// Mitsubishi GX Works2 project: GX_GROUP5   PLC: FX3G

// global labels: Global1
VAR_GLOBAL CONSTANT
  reset1 : INT;
END_VAR
VAR_GLOBAL
  analog_output AT D8282 : INT;
  start_switch AT X007 : BOOL;
  work_light AT Y007 : BOOL;
  emerge_switch AT X005 : BOOL;
  invalid_input AT M7 : BOOL;
  invalid_input_pinuk AT M9 : BOOL;
  petel_begin AT D1102 : REAL;
  petel_current AT D1110 : REAL;
  limon_begin AT D1104 : REAL;
  meyatzev_begin AT D1106 : REAL;
  gummybear_begin AT D1108 : REAL;
  limon_current AT D1112 : REAL;
  meyatzev_current AT D1114 : REAL;
  gummybear_current AT D1116 : REAL;
  start_day AT M0 : BOOL;
  start_icecream AT X001 : BOOL;
  analog_input1 AT D8280 : INT;
  new_analog_input1 AT D1118 : REAL;
END_VAR
VAR_GLOBAL CONSTANT
  convert_input : REAL := 400;
END_VAR
VAR_GLOBAL
  new_analog_input2 AT D1120 : REAL;
  begin_analog_input AT M1 : BOOL;
END_VAR
VAR_GLOBAL CONSTANT
  min_petel : REAL := 280;
  min_limon : REAL := 455;
  min_meyatzev : REAL := 105;
  min_gummybear : REAL := 28;
  const6 : REAL := 6;
  const5 : REAL := 5;
END_VAR
VAR_GLOBAL
  pinuk_ic AT M2 : BOOL;
  regular_ic AT M3 : BOOL;
END_VAR
VAR_GLOBAL CONSTANT
  const385 : REAL := 385;
  const665 : REAL := 665;
  const210 : REAL := 210;
  const70 : REAL := 70;
END_VAR
VAR_GLOBAL
  petelic_container AT D1122 : REAL;
END_VAR
VAR_GLOBAL CONSTANT
  const350 : REAL := 350;
END_VAR
VAR_GLOBAL
  limonic_container AT D1124 : REAL;
END_VAR
VAR_GLOBAL CONSTANT
  const490 : REAL := 490;
END_VAR
VAR_GLOBAL
  finish_regular AT M5 : BOOL;
END_VAR
VAR_GLOBAL CONSTANT
  const560 : REAL := 560;
  const700 : REAL := 700;
END_VAR
VAR_GLOBAL
  finish_pinuk AT M4 : BOOL;
  making_light AT Y000 : BOOL;
  finish_making AT TS1 : BOOL;
  making_time AT TC1 : BOOL;
END_VAR
VAR_GLOBAL CONSTANT
  making_time50 : INT := 50;
  reset_container : REAL;
END_VAR
VAR_GLOBAL
  petel_cooling AT D1126 : REAL;
  limon_cooling AT D1128 : REAL;
  start_cooling AT X002 : BOOL;
  finish_cooling AT Y002 : BOOL;
  sen10 AT X003 : BOOL;
  cooling_timer AT TC2 : BOOL;
END_VAR
VAR_GLOBAL CONSTANT
  cooling_time80 : INT := 80;
END_VAR
VAR_GLOBAL
  container_mix AT D1130 : REAL;
  transfered_to_mix AT M11 : BOOL;
END_VAR
VAR_GLOBAL CONSTANT
  mix_regular_gummybear : REAL := 28;
END_VAR
VAR_GLOBAL
  mix_regular_full AT M12 : BOOL;
  cooling_time AT TS2 : BOOL;
  check AT M101 : BOOL;
  petel_cooling_full AT M10 : BOOL;
  limon_cooling_full AT M17 : BOOL;
END_VAR
VAR_GLOBAL CONSTANT
  mix_pinuk_gummybear : REAL := 70;
END_VAR
VAR_GLOBAL
  mix_pinuk_full AT M13 : BOOL;
  container_mix_total AT D1330 : REAL;
  ready_to_mix AT M15 : BOOL;
END_VAR
VAR_GLOBAL CONSTANT
  regular_mix_time : INT := 30;
END_VAR
VAR_GLOBAL
  mixing_time AT D1132 : INT;
END_VAR
VAR_GLOBAL CONSTANT
  pinuk_mixing_time : INT := 50;
END_VAR
VAR_GLOBAL
  new_mixing_time AT D1134 : INT;
  mixing_time_counter AT TC3 : BOOL;
  finish_counter_mix AT TS3 : BOOL;
  flash_light_mix AT M14 : BOOL;
  flash1 AT TC4 : BOOL;
END_VAR
VAR_GLOBAL CONSTANT
  flash_duration : INT := 5;
END_VAR
VAR_GLOBAL
  timer1 AT TS4 : BOOL;
  light5 AT Y005 : BOOL;
  light6 AT Y006 : BOOL;
  timer2 AT TS5 : BOOL;
  flash2 AT TC5 : BOOL;
  start_packing AT X004 : BOOL;
  first_pack AT CC1 : BOOL;
  counter_pack AT CC2 : BOOL;
  pack_cone AT X000 : BOOL;
END_VAR
VAR_GLOBAL CONSTANT
  counter1 : INT := 1;
END_VAR
VAR_GLOBAL
  outCC2 AT CS2 : BOOL;
  packing AT Y004 : BOOL;
  outCS1 AT CS1 : BOOL;
END_VAR
VAR_GLOBAL CONSTANT
  counter6 : INT := 6;
END_VAR
VAR_GLOBAL
  iteration_help AT M100 : BOOL;
END_VAR
VAR_GLOBAL CONSTANT
  counter7 : INT := 7;
  add_package : INT := 1;
  sec : INT := 10;
END_VAR
VAR_GLOBAL
  amount_packages AT D1200 : REAL;
END_VAR
VAR_GLOBAL CONSTANT
  one_package : REAL := 1;
END_VAR
VAR_GLOBAL
  check2 AT M102 : BOOL;
  finish_making_light AT M200 : BOOL;
  finish_cooling_light AT M201 : BOOL;
END_VAR
VAR_GLOBAL CONSTANT
  const40 : REAL := 40;
END_VAR
VAR_GLOBAL
  new_amount_package AT D1136 : REAL;
END_VAR

// task Task_01 (event TRUE, interval 0, priority 31): POU_01

PROGRAM POU_01
(* structured ladder/FBD written out as ST: instructions are called as NAME(EN, inputs, outputs); _pN, _eN, _tN stand for wires *)
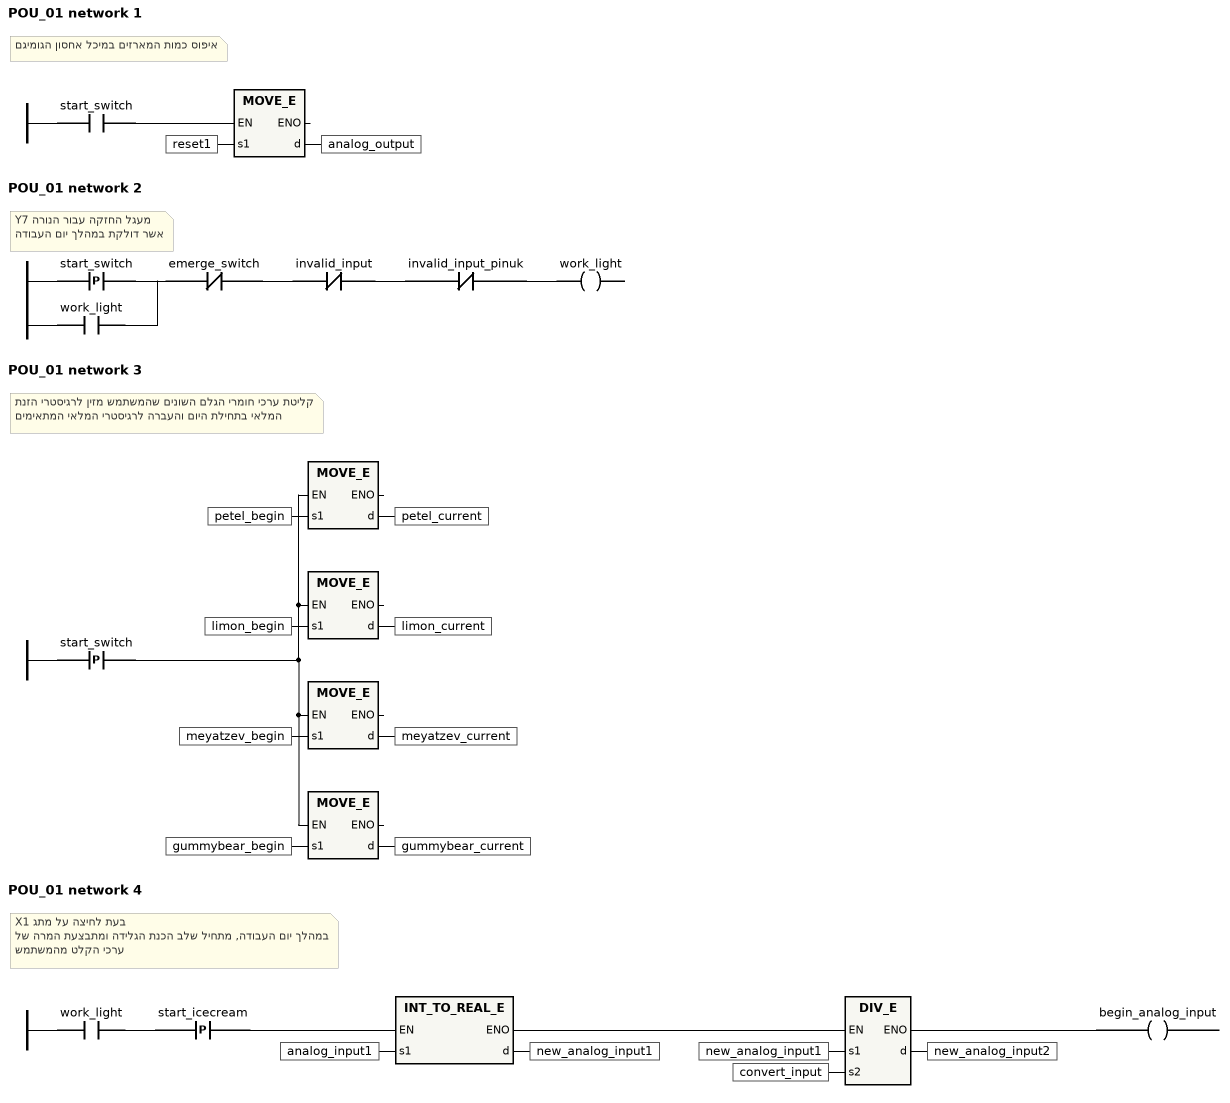
(* network 1 *)
(* איפוס כמות המארזים במיכל אחסון הגומיגם *)
MOVE_E(start_switch, reset1, analog_output);
(* network 2 *)
(* מעגל החזקה עבור הנורה Y7 /  אשר דולקת במהלך יום העבודה *)
work_light := (((LDP(TRUE, start_switch) OR work_light) AND NOT emerge_switch) AND NOT invalid_input) AND NOT invalid_input_pinuk;
(* network 3 *)
(* קליטת ערכי חומרי הגלם השונים שהמשתמש מזין לרגיסטרי הזנת המלאי בתחילת היום והעברה לרגיסטרי המלאי המתאימים *)
_p1 := LDP(TRUE, start_switch);
MOVE_E(_p1, petel_begin, petel_current);
MOVE_E(_p1, limon_begin, limon_current);
MOVE_E(_p1, meyatzev_begin, meyatzev_current);
MOVE_E(_p1, gummybear_begin, gummybear_current);
(* network 4 *)
(* בעת לחיצה על מתג X1  / במהלך יום העבודה, מתחיל שלב הכנת הגלידה ומתבצעת המרה של ערכי הקלט מהמשתמש *)
_e1 := INT_TO_REAL_E(work_light AND LDP(TRUE, start_icecream), analog_input1, new_analog_input1);
_e2 := DIV_E(_e1, new_analog_input1, convert_input, new_analog_input2);
begin_analog_input := _e2;
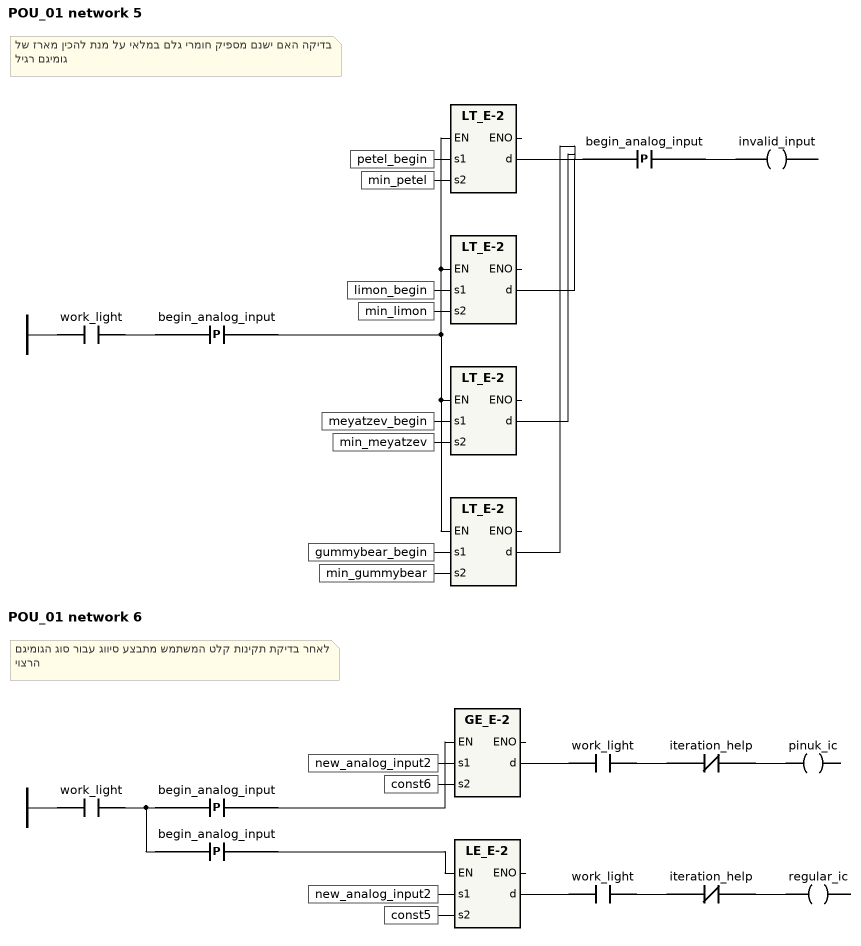
(* network 5 *)
(* בדיקה האם ישנם מספיק חומרי גלם במלאי על מנת להכין מארז של גומיגם רגיל *)
_p1 := work_light AND LDP(TRUE, begin_analog_input);
LT_E(_p1, petel_begin, min_petel, _t2);
LT_E(_p1, limon_begin, min_limon, _t3);
LT_E(_p1, meyatzev_begin, min_meyatzev, _t4);
LT_E(_p1, gummybear_begin, min_gummybear, _t5);
invalid_input := (_t2 OR _t3 OR _t4 OR _t5) AND LDP(TRUE, begin_analog_input);
(* network 6 *)
(* לאחר בדיקת תקינות קלט המשתמש מתבצע סיווג עבור סוג הגומיגם הרצוי *)
GE_E(work_light AND LDP(TRUE, begin_analog_input), new_analog_input2, const6, _t1);
pinuk_ic := _t1 AND work_light AND NOT iteration_help;
LE_E(work_light AND LDP(TRUE, begin_analog_input), new_analog_input2, const5, _t2);
regular_ic := _t2 AND work_light AND NOT iteration_help;
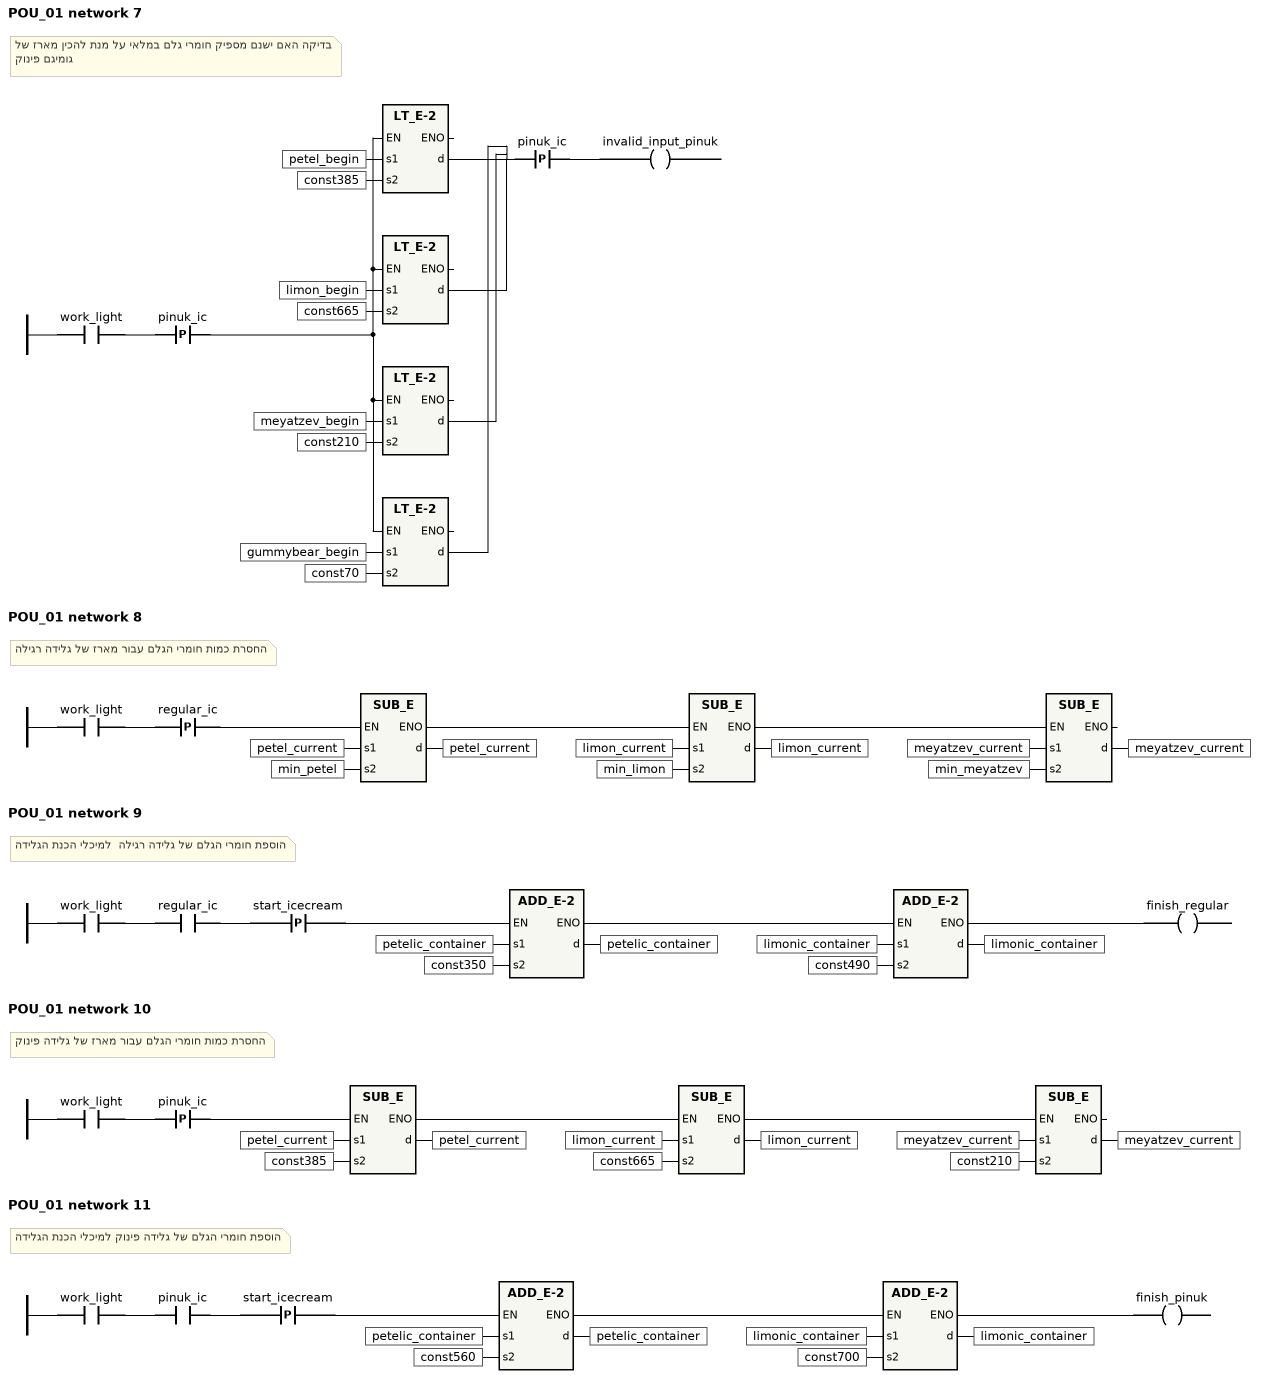
(* network 7 *)
(* בדיקה האם ישנם מספיק חומרי גלם במלאי על מנת להכין מארז של גומיגם פינוק *)
_p1 := work_light AND LDP(TRUE, pinuk_ic);
LT_E(_p1, petel_begin, const385, _t2);
LT_E(_p1, limon_begin, const665, _t3);
LT_E(_p1, meyatzev_begin, const210, _t4);
LT_E(_p1, gummybear_begin, const70, _t5);
invalid_input_pinuk := (_t2 OR _t3 OR _t4 OR _t5) AND LDP(TRUE, pinuk_ic);
(* network 8 *)
(* החסרת כמות חומרי הגלם עבור מארז של גלידה רגילה *)
_e1 := SUB_E(work_light AND LDP(TRUE, regular_ic), petel_current, min_petel, petel_current);
_e2 := SUB_E(_e1, limon_current, min_limon, limon_current);
SUB_E(_e2, meyatzev_current, min_meyatzev, meyatzev_current);
(* network 9 *)
(* הוספת חומרי הגלם של גלידה רגילה  למיכלי הכנת הגלידה *)
_e1 := ADD_E(work_light AND regular_ic AND LDP(TRUE, start_icecream), petelic_container, const350, petelic_container);
_e2 := ADD_E(_e1, limonic_container, const490, limonic_container);
finish_regular := _e2;
(* network 10 *)
(* החסרת כמות חומרי הגלם עבור מארז של גלידה פינוק *)
_e1 := SUB_E(work_light AND LDP(TRUE, pinuk_ic), petel_current, const385, petel_current);
_e2 := SUB_E(_e1, limon_current, const665, limon_current);
SUB_E(_e2, meyatzev_current, const210, meyatzev_current);
(* network 11 *)
(* הוספת חומרי הגלם של גלידה פינוק למיכלי הכנת הגלידה *)
_e1 := ADD_E(work_light AND pinuk_ic AND LDP(TRUE, start_icecream), petelic_container, const560, petelic_container);
_e2 := ADD_E(_e1, limonic_container, const700, limonic_container);
finish_pinuk := _e2;
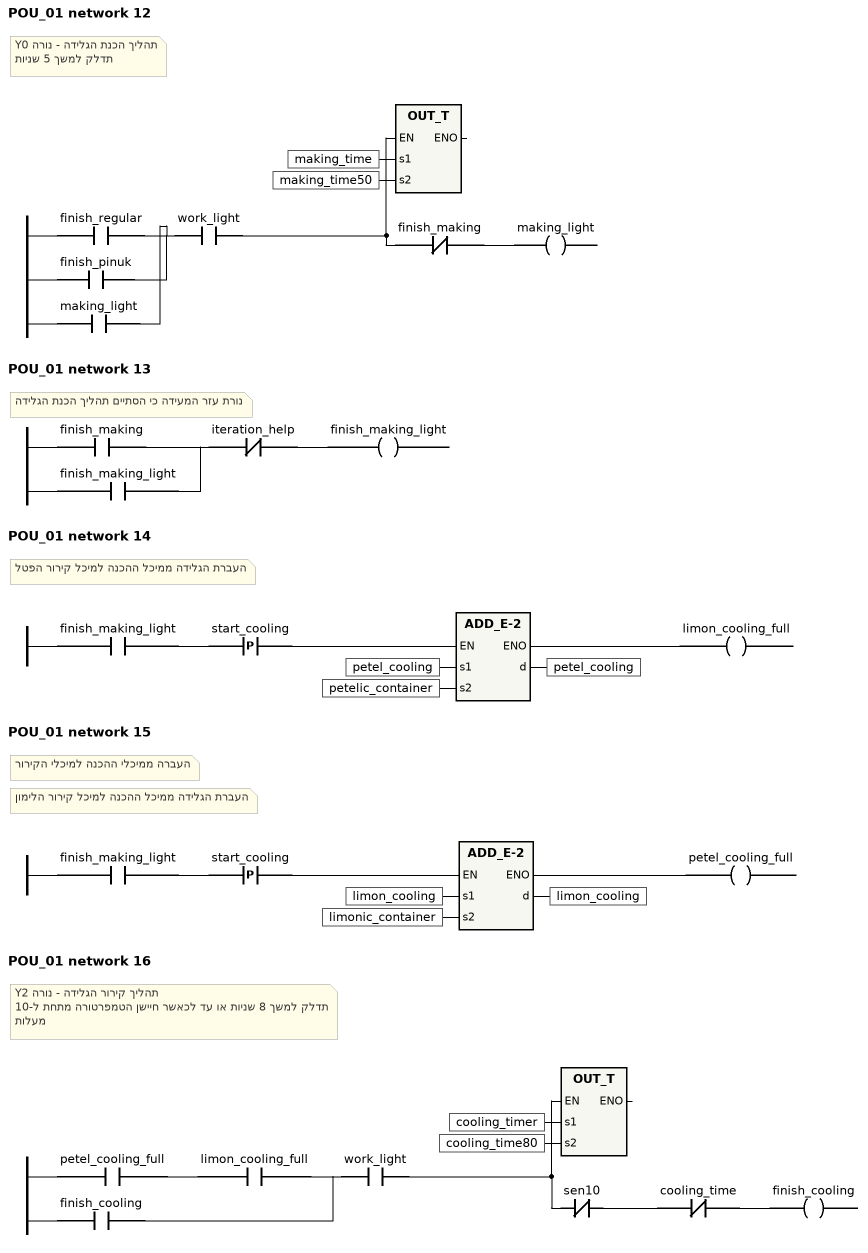
(* network 12 *)
(* תהליך הכנת הגלידה - נורה Y0 /  תדלק למשך 5 שניות *)
_p1 := (finish_regular OR finish_pinuk OR making_light) AND work_light;
OUT_T(_p1, making_time, making_time50);
making_light := _p1 AND NOT finish_making;
(* network 13 *)
(* נורת עזר המעידה כי הסתיים תהליך הכנת הגלידה *)
finish_making_light := (finish_making OR finish_making_light) AND NOT iteration_help;
(* network 14 *)
(* העברת הגלידה ממיכל ההכנה למיכל קירור הפטל *)
_e1 := ADD_E(finish_making_light AND LDP(TRUE, start_cooling), petel_cooling, petelic_container, petel_cooling);
limon_cooling_full := _e1;
(* network 15 *)
(* העברה ממיכלי ההכנה למיכלי הקירור *)
(* העברת הגלידה ממיכל ההכנה למיכל קירור הלימון *)
_e1 := ADD_E(finish_making_light AND LDP(TRUE, start_cooling), limon_cooling, limonic_container, limon_cooling);
petel_cooling_full := _e1;
(* network 16 *)
(* תהליך קירור הגלידה - נורה Y2 /  תדלק למשך 8 שניות או עד לכאשר חיישן הטמפרטורה מתחת ל-10 מעלות *)
_p1 := ((petel_cooling_full AND limon_cooling_full) OR finish_cooling) AND work_light;
OUT_T(_p1, cooling_timer, cooling_time80);
finish_cooling := _p1 AND NOT sen10 AND NOT cooling_time;
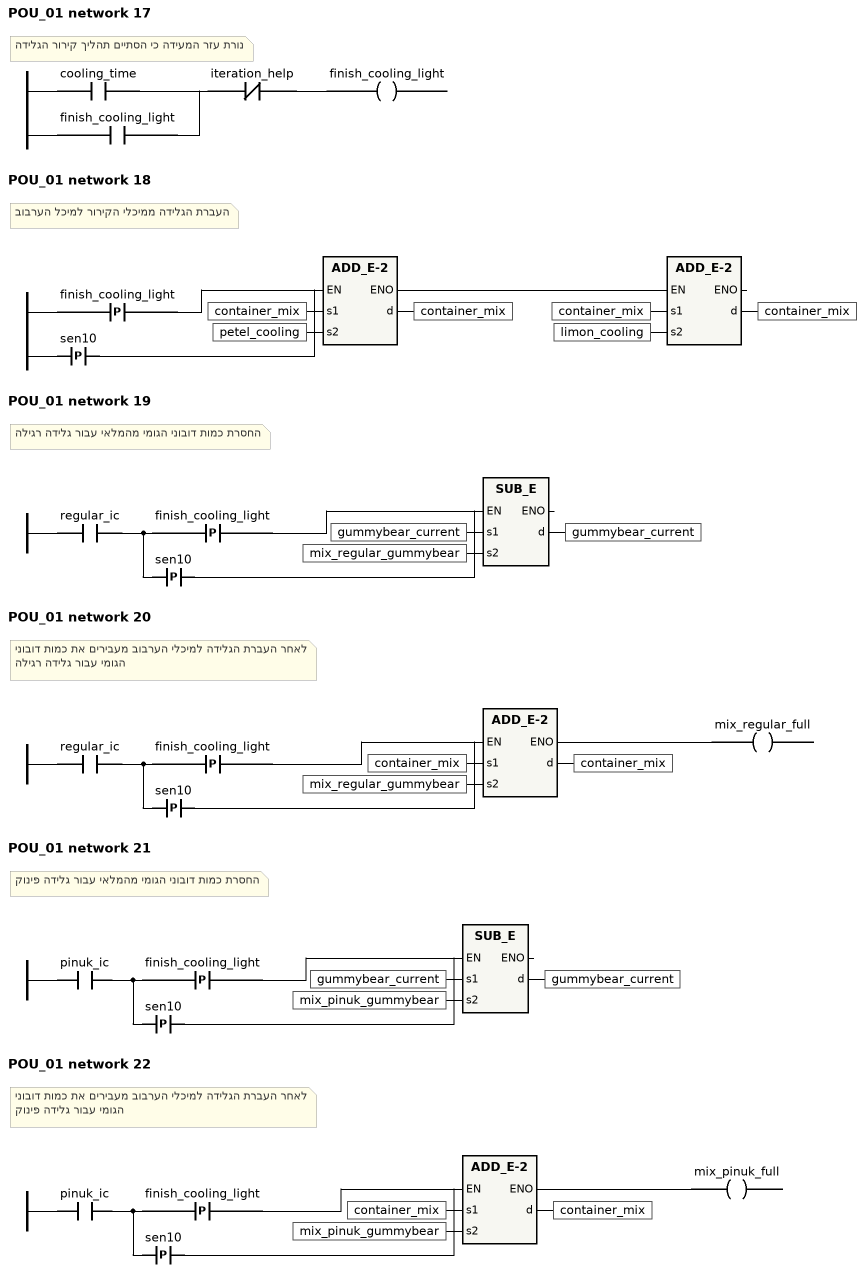
(* network 17 *)
(* נורת עזר המעידה כי הסתיים תהליך קירור הגלידה *)
finish_cooling_light := (cooling_time OR finish_cooling_light) AND NOT iteration_help;
(* network 18 *)
(* העברת הגלידה ממיכלי הקירור למיכל הערבוב *)
_e1 := ADD_E(LDP(TRUE, finish_cooling_light) OR LDP(TRUE, sen10), container_mix, petel_cooling, container_mix);
ADD_E(_e1, container_mix, limon_cooling, container_mix);
(* network 19 *)
(* החסרת כמות דובוני הגומי מהמלאי עבור גלידה רגילה *)
SUB_E((regular_ic AND LDP(TRUE, finish_cooling_light)) OR (regular_ic AND LDP(TRUE, sen10)), gummybear_current, mix_regular_gummybear, gummybear_current);
(* network 20 *)
(* לאחר העברת הגלידה למיכלי הערבוב מעבירים את כמות דובוני הגומי עבור גלידה רגילה *)
_e1 := ADD_E((regular_ic AND LDP(TRUE, finish_cooling_light)) OR (regular_ic AND LDP(TRUE, sen10)), container_mix, mix_regular_gummybear, container_mix);
mix_regular_full := _e1;
(* network 21 *)
(* החסרת כמות דובוני הגומי מהמלאי עבור גלידה פינוק *)
SUB_E((pinuk_ic AND LDP(TRUE, finish_cooling_light)) OR (pinuk_ic AND LDP(TRUE, sen10)), gummybear_current, mix_pinuk_gummybear, gummybear_current);
(* network 22 *)
(* לאחר העברת הגלידה למיכלי הערבוב מעבירים את כמות דובוני הגומי עבור גלידה פינוק *)
_e1 := ADD_E((pinuk_ic AND LDP(TRUE, finish_cooling_light)) OR (pinuk_ic AND LDP(TRUE, sen10)), container_mix, mix_pinuk_gummybear, container_mix);
mix_pinuk_full := _e1;
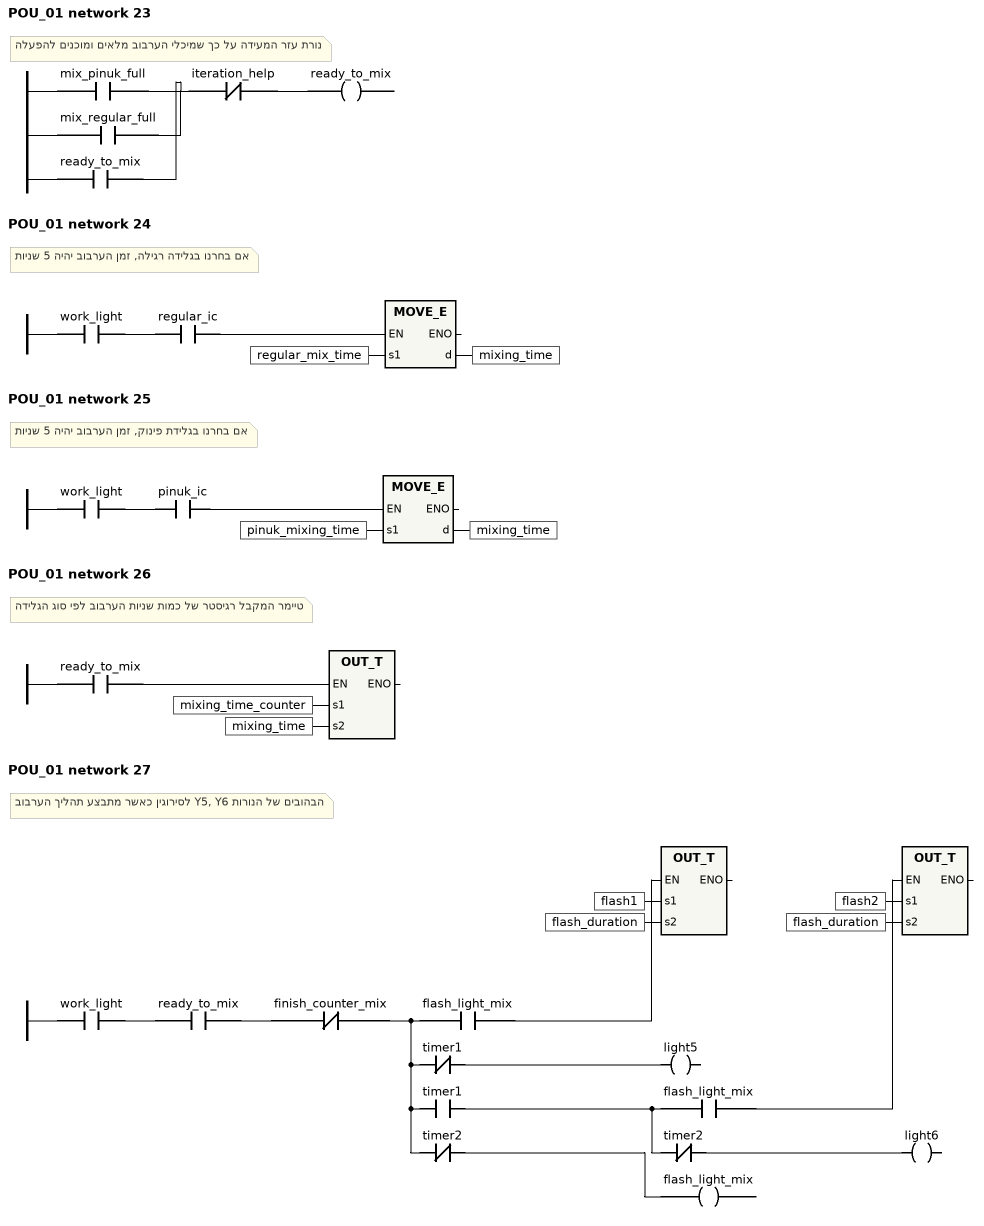
(* network 23 *)
(* נורת עזר המעידה על כך שמיכלי הערבוב מלאים ומוכנים להפעלה *)
ready_to_mix := (mix_pinuk_full OR mix_regular_full OR ready_to_mix) AND NOT iteration_help;
(* network 24 *)
(* אם בחרנו בגלידה רגילה, זמן הערבוב יהיה 5 שניות *)
MOVE_E(work_light AND regular_ic, regular_mix_time, mixing_time);
(* network 25 *)
(* אם בחרנו בגלידת פינוק, זמן הערבוב יהיה 5 שניות *)
MOVE_E(work_light AND pinuk_ic, pinuk_mixing_time, mixing_time);
(* network 26 *)
(* טיימר המקבל רגיסטר של כמות שניות הערבוב לפי סוג הגלידה *)
OUT_T(ready_to_mix, mixing_time_counter, mixing_time);
(* network 27 *)
(* הבהובים של הנורות Y5, Y6 לסירוגין כאשר מתבצע תהליך הערבוב *)
_p1 := work_light AND ready_to_mix AND NOT finish_counter_mix;
OUT_T(_p1 AND flash_light_mix, flash1, flash_duration);
light5 := _p1 AND NOT timer1;
_p2 := _p1 AND timer1;
OUT_T(_p2 AND flash_light_mix, flash2, flash_duration);
light6 := _p2 AND NOT timer2;
flash_light_mix := _p1 AND NOT timer2;
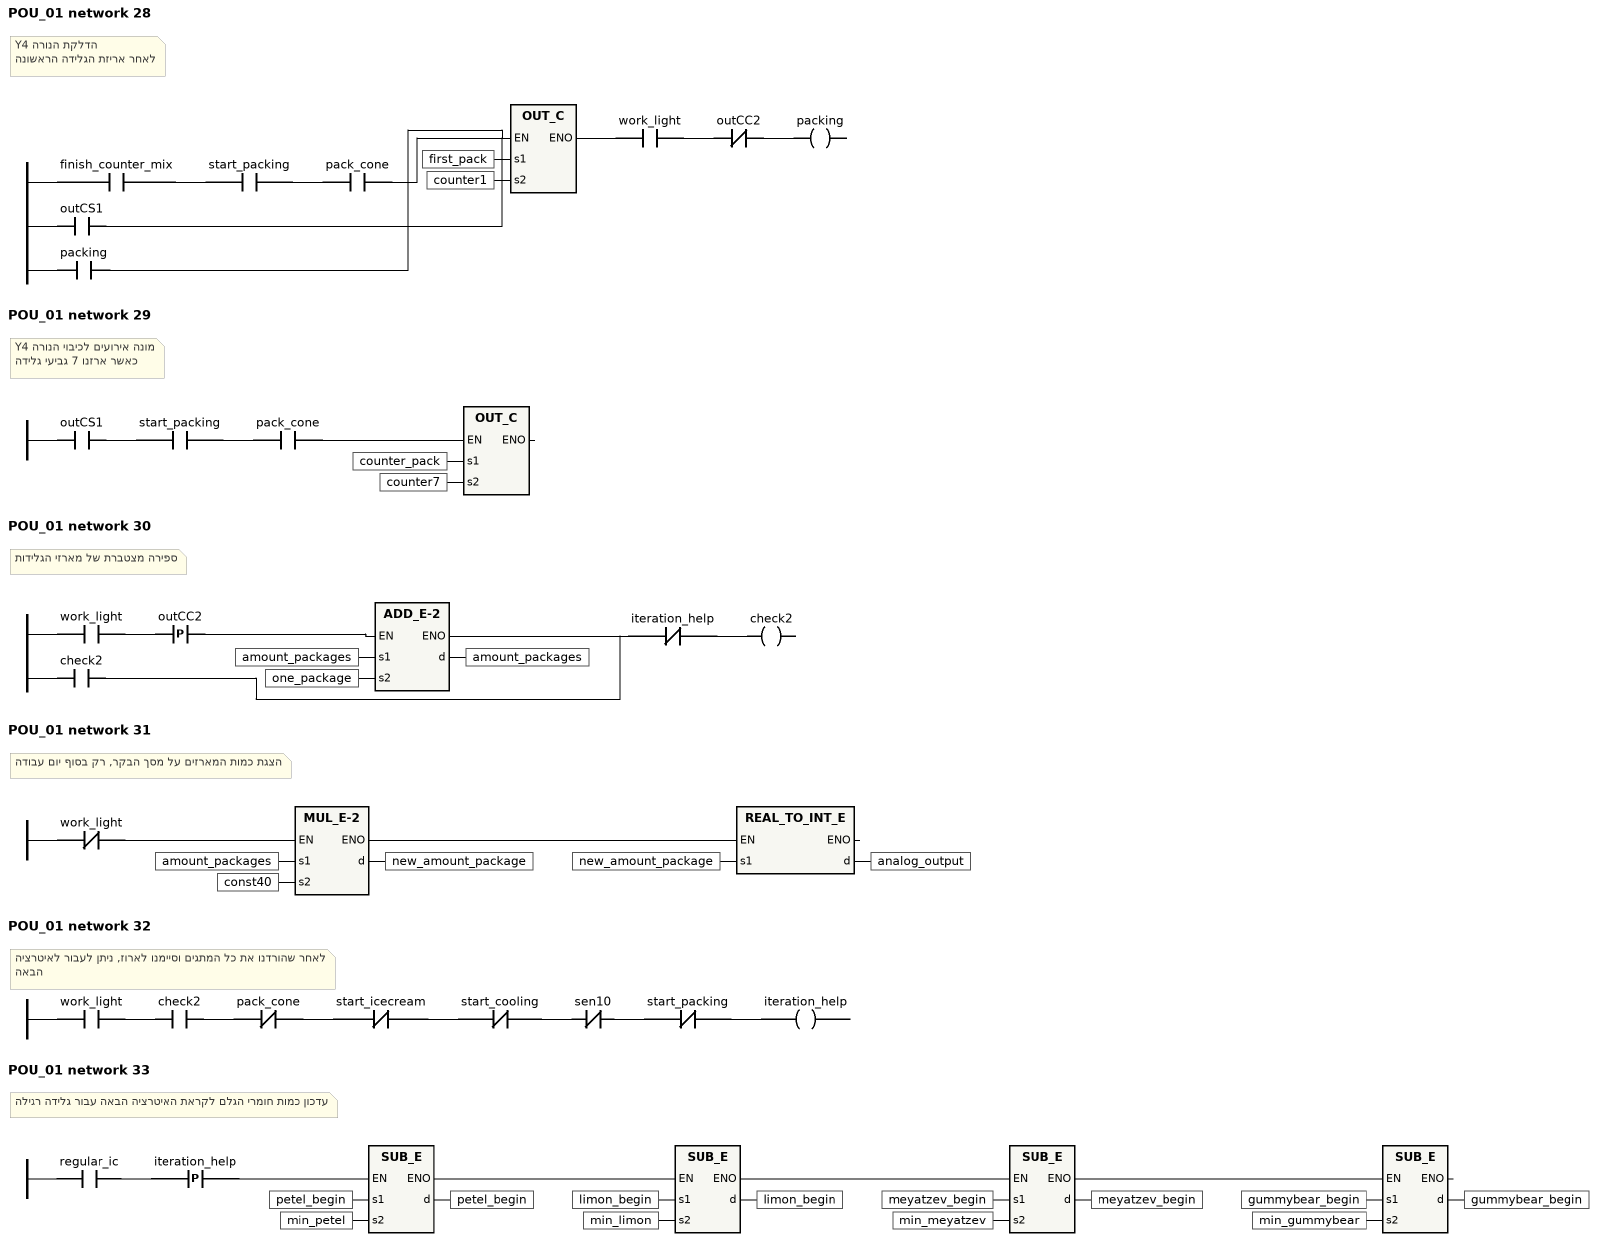
(* network 28 *)
(* הדלקת הנורה Y4 / לאחר אריזת הגלידה הראשונה *)
_e1 := OUT_C((finish_counter_mix AND start_packing AND pack_cone) OR outCS1 OR packing, first_pack, counter1);
packing := _e1 AND work_light AND NOT outCC2;
(* network 29 *)
(* מונה אירועים לכיבוי הנורה Y4  / כאשר ארזנו 7 גביעי גלידה *)
OUT_C(outCS1 AND start_packing AND pack_cone, counter_pack, counter7);
(* network 30 *)
(* ספירה מצטברת של מארזי הגלידות *)
_e1 := ADD_E(work_light AND LDP(TRUE, outCC2), amount_packages, one_package, amount_packages);
check2 := (_e1 OR check2) AND NOT iteration_help;
(* network 31 *)
(* הצגת כמות המארזים על מסך הבקר, רק בסוף יום עבודה *)
_e1 := MUL_E(NOT work_light, amount_packages, const40, new_amount_package);
REAL_TO_INT_E(_e1, new_amount_package, analog_output);
(* network 32 *)
(* לאחר שהורדנו את כל המתגים וסיימנו לארוז, ניתן לעבור לאיטרציה הבאה *)
iteration_help := work_light AND check2 AND NOT pack_cone AND NOT start_icecream AND NOT start_cooling AND NOT sen10 AND NOT start_packing;
(* network 33 *)
(* עדכון כמות חומרי הגלם לקראת האיטרציה הבאה עבור גלידה רגילה *)
_e1 := SUB_E(regular_ic AND LDP(TRUE, iteration_help), petel_begin, min_petel, petel_begin);
_e2 := SUB_E(_e1, limon_begin, min_limon, limon_begin);
_e3 := SUB_E(_e2, meyatzev_begin, min_meyatzev, meyatzev_begin);
SUB_E(_e3, gummybear_begin, min_gummybear, gummybear_begin);
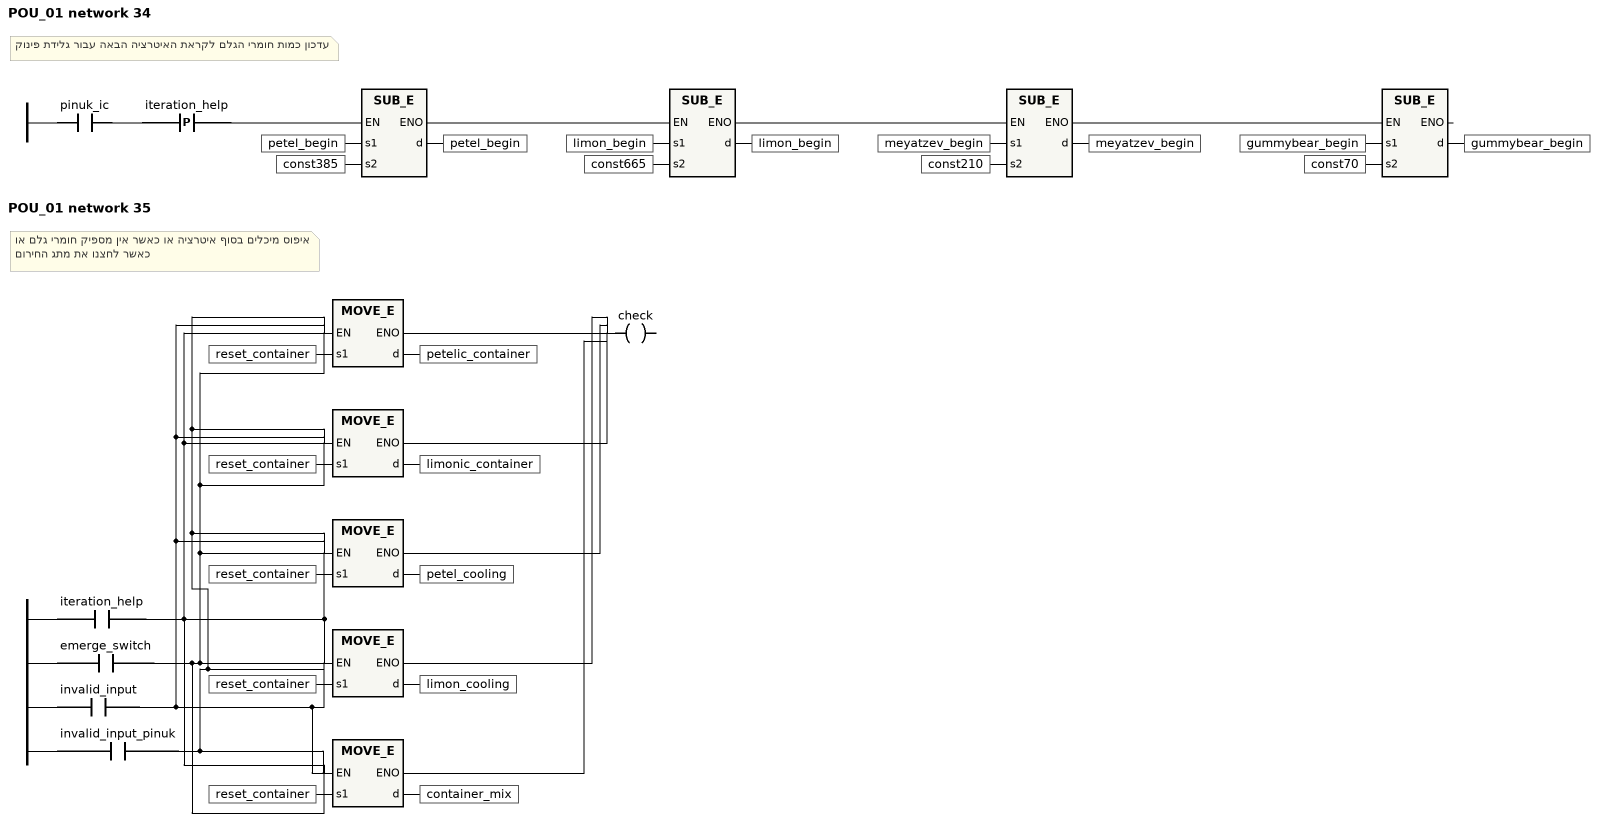
(* network 34 *)
(* עדכון כמות חומרי הגלם לקראת האיטרציה הבאה עבור גלידת פינוק *)
_e1 := SUB_E(pinuk_ic AND LDP(TRUE, iteration_help), petel_begin, const385, petel_begin);
_e2 := SUB_E(_e1, limon_begin, const665, limon_begin);
_e3 := SUB_E(_e2, meyatzev_begin, const210, meyatzev_begin);
SUB_E(_e3, gummybear_begin, const70, gummybear_begin);
(* network 35 *)
(* איפוס מיכלים בסוף איטרציה או כאשר אין מספיק חומרי גלם או כאשר לחצנו את מתג החירום *)
_p1 := iteration_help OR emerge_switch OR invalid_input OR invalid_input_pinuk;
_e2 := MOVE_E(_p1, reset_container, petelic_container);
_e3 := MOVE_E(_p1, reset_container, limonic_container);
_e4 := MOVE_E(_p1, reset_container, petel_cooling);
_e5 := MOVE_E(_p1, reset_container, limon_cooling);
_e6 := MOVE_E(_p1, reset_container, container_mix);
check := _e2 OR _e3 OR _e4 OR _e5 OR _e6;
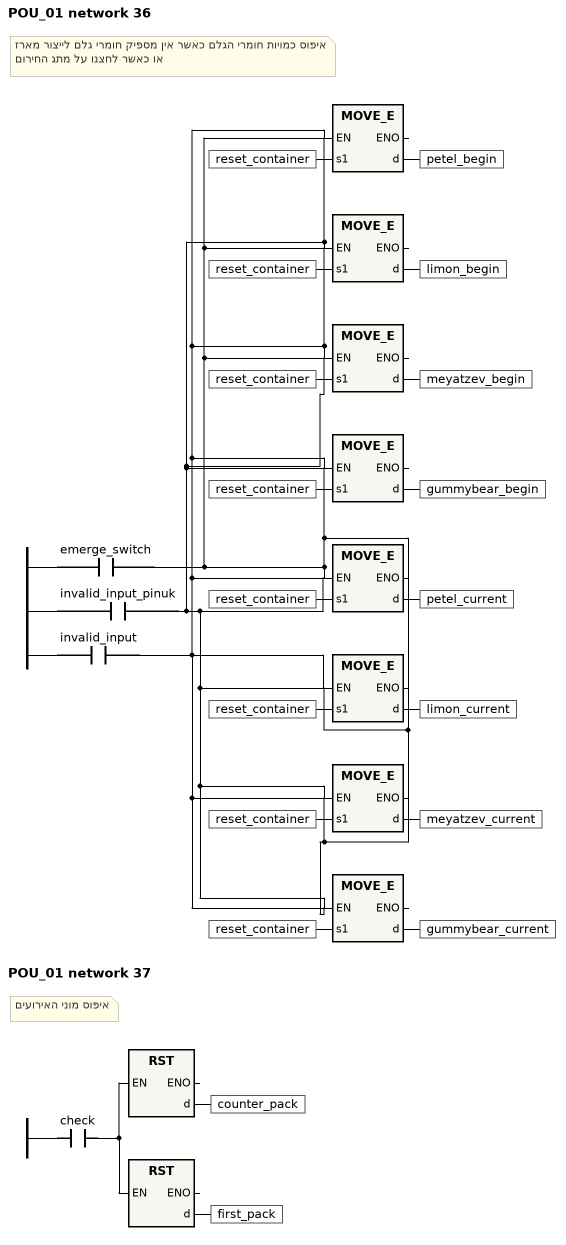
(* network 36 *)
(* איפוס כמויות חומרי הגלם כאשר אין מספיק חומרי גלם לייצור מארז או כאשר לחצנו על מתג החירום *)
_p1 := emerge_switch OR invalid_input_pinuk OR invalid_input;
MOVE_E(_p1, reset_container, petel_begin);
MOVE_E(_p1, reset_container, limon_begin);
MOVE_E(_p1, reset_container, meyatzev_begin);
MOVE_E(_p1, reset_container, gummybear_begin);
MOVE_E(_p1, reset_container, petel_current);
MOVE_E(_p1, reset_container, limon_current);
MOVE_E(_p1, reset_container, meyatzev_current);
MOVE_E(_p1, reset_container, gummybear_current);
(* network 37 *)
(* איפוס מוני האירועים *)
RST(check, counter_pack);
RST(check, first_pack);
END_PROGRAM
